TYPE LogConfig :
STRUCT
	LogFileConfigPath : STRING;
	HeaderNodeXml : STRING;
	LogFilePath : STRING;
	AddLogsConsole : BOOL;
END_STRUCT
END_TYPE

(* stored: Version 1.1.0.1, ProductVersion 3.1.4024.3
   DUT LogConfig: Id {dbe18cf8-74ff-4912-8940-0b842e62dc21} *)
